(*
    The sensor contract every miniload module reads a discrete signal through.
    A consumer holds an I_DigitalInput and asks it what the signal MEANS -
    settled, in field polarity - never what the wire is doing right now. The
    consumer does not cycle the sensor; whoever owns the instance does.

    DebounceTime is symmetric: it gates both the rising and the falling
    transition, so a chattering photo-eye cannot make Active flicker in either
    direction.

    TimeActive / TimeInactive measure the CURRENT unbroken stretch in that
    state and reset on every settled transition. They answer "how long has
    this been so", not "how long in total", which is what a blocked-conveyor
    or missing-container diagnostic needs.

    Simulation is the seam a mock hangs off: with Simulation set, SimulatedInput
    replaces the field bit and everything downstream - polarity, debounce,
    elapsed time - behaves exactly as it does on real hardware.
*)
INTERFACE I_DigitalInput

// The settled, polarity-corrected signal.
PROPERTY Active : BOOL
GET
END_GET
END_PROPERTY

// How long a level must hold before it is allowed to move Active, in
// both directions. Zero means no filtering at all.
PROPERTY DebounceTime : TIME
GET
END_GET
SET
END_SET
END_PROPERTY

// TRUE for a normally closed sensor: the wire level is negated before
// anything else looks at it.
PROPERTY Inverted : BOOL
GET
END_GET
SET
END_SET
END_PROPERTY

// Selects SimulatedInput over the field bit.
PROPERTY Simulation : BOOL
GET
END_GET
SET
END_SET
END_PROPERTY

// The stand-in level, read only while Simulation is set. Writing it with
// Simulation clear changes nothing, so a test may arm it up front.
PROPERTY SimulatedInput : BOOL
GET
END_GET
SET
END_SET
END_PROPERTY

// Length of the current unbroken active stretch; zero whenever inactive.
PROPERTY TimeActive : TIME
GET
END_GET
END_PROPERTY

// Length of the current unbroken inactive stretch; zero whenever active.
PROPERTY TimeInactive : TIME
GET
END_GET
END_PROPERTY

END_INTERFACE

(* stored: Version 1.1.0.1, ProductVersion 3.1.4026.18
   Itf I_DigitalInput: Id {5e4501d0-0001-4d19-9a41-000000000001}
   Property Active: Id {5e4501d0-0001-4d19-9a41-000000000002}
   Get Get: Id {5e4501d0-0001-4d19-9a41-000000000003}
   Property DebounceTime: Id {5e4501d0-0001-4d19-9a41-000000000004}
   Get Get: Id {5e4501d0-0001-4d19-9a41-000000000005}
   Set Set: Id {5e4501d0-0001-4d19-9a41-000000000006}
   Property Inverted: Id {5e4501d0-0001-4d19-9a41-000000000007}
   Get Get: Id {5e4501d0-0001-4d19-9a41-000000000008}
   Set Set: Id {5e4501d0-0001-4d19-9a41-000000000009}
   Property Simulation: Id {5e4501d0-0001-4d19-9a41-00000000000a}
   Get Get: Id {5e4501d0-0001-4d19-9a41-00000000000b}
   Set Set: Id {5e4501d0-0001-4d19-9a41-00000000000c}
   Property SimulatedInput: Id {5e4501d0-0001-4d19-9a41-00000000000d}
   Get Get: Id {5e4501d0-0001-4d19-9a41-00000000000e}
   Set Set: Id {5e4501d0-0001-4d19-9a41-00000000000f}
   Property TimeActive: Id {5e4501d0-0001-4d19-9a41-000000000010}
   Get Get: Id {5e4501d0-0001-4d19-9a41-000000000011}
   Property TimeInactive: Id {5e4501d0-0001-4d19-9a41-000000000012}
   Get Get: Id {5e4501d0-0001-4d19-9a41-000000000013} *)
